(* CODESYS project SingleElevator.project

Project tree, tasks and I/O mapping:
  Device : CODESYS Control Win V3, CODESYS, version 3.5.21.30
    application Application
      libraries: Standard, 3.5.18.0 (System)
      task MainTask (cyclic, interval t#20ms, priority 1) calls Simulation, GA_collector, PLC_Program
      task VISU_TASK (cyclic, interval 100 ms, priority 31) calls VisuElems.Visu_Prg
      global variables GVL
      visualisation Visualization
      program Simulation [ST]
      data type State_FB
      data type DoWhats
      data type Action_s
      program GA_collector [FBD]
      program PLC_Program [SFC]: _astart_led_active, _ainitialize_active, _ainitialize_exit, _ago_destination_active, _ago_destination_exit, _adoors_init_active, _adoors_open_active, _adoors_init_exit, _adoors_open_exit, _adoors_open1_active, _adoors_open1_exit, _adoors_closing_exit_1, _adoors_closing_active_1, _afault_block_entry
      function block Door_opener [SFC]: _aInit_active, _aReady_active, _aReady_exit, _aopening_door_active, _aClosing_door_active, _aopening_door_exit, _afinish_closing_exit, _aopen_again_active, _aopen_again_exit, _aSetDone_active, _aSetDone_exit, _afinish_closing_active
      function block motor [SFC]: _aReady_active, _aReady_exit, _aInit_active, _adescent_active, _aascent_active, _aSetDone_active, _adeck_fault_exit, _aSetDone_exit, _amove1_active, _await1s_entry, _amove1_exit, _aSetDone1_exit, _aSetDone1_active, _astop_motor_entry, _aset_vel_active, _adummy1_entry, _aRamp_Fault_active, _aSetDone2_entry, _aSetDone2_active, _aSetDone2_exit, _aspeed_inverter_entry, _aSetDone4_active, _aSetDone4_exit, _aascent_exit, _acurrent_add_entry, _aRamp_Fault_entry
      function block LEDs [SFC]: _aAssignCalls_active, _aAssignCalls_active_1, _aInit_active, _aReady_active_1, _aReady_exit_1
  text list GlobalTextList
  function block LEDs [SFC]: _aAssignCalls_active, _aAssignCalls_active_1, _aInit_active, _aReady_active_1, _aReady_exit_1
*)

// Device/Application/State_FB
//{attribute 'qualified_only'}
//{attribute 'strict'}// if we don't comment we need to use the nameofthetype.chosentype
TYPE State_FB :
(
	S_Init := 0,// never call a variable with the same name of a step
	S_Ready:=1,
	S_Busy:=2,
	S_Faulty:=3
	// we'll use the strings so it is more readable
);
END_TYPE

// Device/Application/DoWhats
//{attribute 'qualified_only'}
//{attribute 'strict'}
TYPE DoWhats :
(
	Gotodestination := 0,
	Initialize :=1,
	door_closing:=2,
	door_opening:=3
);
END_TYPE

// Device/Application/Action_s
//{attribute 'qualified_only'}
//{attribute 'strict'}
TYPE Action_s :
(
	start_action:=0,
	Wait_comp:=1,
	setopOK:=2
);
END_TYPE

// Device/Application/GVL
{attribute 'qualified_only'}
VAR_GLOBAL
(* Elevator managing variables*)
	Open: BOOL;				(* Sensor: the door is fully open*)
	Closed: BOOL;			(* Sensor: the door is fully closed*)
	LimitDown: BOOL;		(* Sensor: lower limit sensor, if TRUE the lift has reached the lower limit*)
	LimitUp: BOOL;			(* Sensor: upper limit sensor, if TRUE the lift has reached the upper limit*)
	DeckSensor: BOOL;		(* Sensor: if TRUE the cab is in proximity of a deck*)
	RampSensor: BOOL;		(* Sensor: if TRUE the cab is in proximity of a ramp*)
	Presence :BOOL; 		(* Sensor: if TRUE something blocks the door photocell*)
	

	Closing: BOOL;			(* Actuator: if TRUE the door starts closing*)
	Opening: BOOL;			(* Actuator: the door starts opening*)
	Motor_on: BOOL;			(* Actuator: if TRUE the lift pulley motor start moving*)
	Up: BOOL;				(* Actuator parameter: if TRUE the lift moves upward, downward otherwise*)
	Vel: BOOL;				(* Actuator parameter: motor speed, if TRUE high speed, low speed otherwise*)


	Current: INT;  			(* Visualization: variable used to storage the current deck*)
    Destination: INT;		(* Visualization: variable used to storage the the destination deck*)
	

	InitialDeck: INT := 1;	(* Only for simulation: variable used to define the initial deck*)
	InitCycle: BOOL := FALSE;(* Only for simulation: used to execute the instruction at the first cycle*)
	Height: INT;			(* Only for simulation: elevator height*)
	DeckRest: INT;        	(* Only for simulation: division rest for generating deck sensor*)
	Memory: INT;
	RampRest: INT;			(* Only for simulation: division rest for generating the ramp position*)
	MemoryR: INT;
	Door: INT;				(* Only for simulation: to visualize the closing of the door*)
	Displacement: INT;		(* Only for simulation: lift displacement, dependent on the motor speed*)

 (*Inputs: internal panel variables*)
	PG: BOOL;
	P1: BOOL;
	P2: BOOL;
	P3: BOOL;
	P4: BOOL;
	P5: BOOL;
	P6: BOOL;
	P7: BOOL;

(*Visualization: internal panel variables used to turn on the LED*)
	PGVis: BOOL;
	P1Vis: BOOL;
	P2Vis: BOOL;
	P3Vis: BOOL;
	P4Vis: BOOL;
	P5Vis: BOOL;
	P6Vis: BOOL;
	P7Vis: BOOL;

(*Inputs: external panel variables*)
	UpDeckG: BOOL;
	UpDeck1: BOOL;
	UpDeck2: BOOL;
	UpDeck3: BOOL;
	UpDeck4: BOOL;
	UpDeck5: BOOL;
	UpDeck6: BOOL;
	DownDeck7: BOOL;
	DownDeck6: BOOL;
	DownDeck5: BOOL;
	DownDeck4: BOOL;
	DownDeck3: BOOL;
	DownDeck2: BOOL;
	DownDeck1: BOOL;

(*Visualization: external panel variables used to turn on the LED*)
	UpDeckGVis: BOOL;
	UpDeck1Vis: BOOL;
	UpDeck2Vis: BOOL;
	UpDeck3Vis: BOOL;
	UpDeck4Vis: BOOL;
	UpDeck5Vis: BOOL;
	UpDeck6Vis: BOOL;
	DownDeck7Vis: BOOL;
	DownDeck6Vis: BOOL;
	DownDeck5Vis: BOOL;
	DownDeck4Vis: BOOL;
	DownDeck3Vis: BOOL;
	DownDeck2Vis: BOOL;
	DownDeck1Vis: BOOL;

(*Only for simulation: variables used to simulate the fault on deck sensor*)
	SensorG: BOOL;				(* if TRUE the magnetic information for deck G is lost and the deck sensor cannot become TRUE*)
	Sensor1: BOOL;				(* if TRUE the magnetic information for deck 1 is lost and the deck sensor cannot become TRUE*)
	Sensor2: BOOL;
	Sensor3: BOOL;
	Sensor4: BOOL;
	Sensor5: BOOL;
	Sensor6: BOOL;
	Sensor7: BOOL;
	FaultSensorAlarm: BOOL; 	(* Visulaization: if TRUE alerts the user of a deck sensor fault*)

(*Only for simulation: variables used to simulate the fault on ramp sensor*)
	RampGUp: BOOL;
	Ramp1Down: BOOL;
	Ramp1Up:BOOL;
	Ramp2Down: BOOL;
	Ramp2Up:BOOL;
	Ramp3Down: BOOL;
	Ramp3Up:BOOL;
	Ramp4Down: BOOL;
	Ramp4Up:BOOL;
	Ramp5Down: BOOL;
	Ramp5Up:BOOL;
	Ramp6Down: BOOL;
	Ramp6Up:BOOL;
	Ramp7Down: BOOL;
	FaultRampAlarm: BOOL; 		(* Visulaization: if TRUE alerts the user of a ramp sensor fault*)
	SensorGOK: BOOL;
	Sensor1OK: BOOL;
	Sensor2OK: BOOL;
	Sensor6OK: BOOL;
	Sensor3OK: BOOL;
	Sensor4OK: BOOL;
	Sensor5OK: BOOL;
	Sensor7OK: BOOL;
	RampGUpOK: BOOL;
	Ramp1DownOK: BOOL;
	Ramp1UpOK: BOOL;
	Ramp2DownOK: BOOL;
	Ramp2UpOK: BOOL;
	Ramp3DownOK: BOOL;
	Ramp3UpOK: BOOL;
	Ramp4DownOK: BOOL;
	Ramp4UpOK: BOOL;
	Ramp5DownOK: BOOL;
	Ramp5UpOK: BOOL;
	Ramp6DownOK: BOOL;
	Ramp6UpOK: BOOL;
	Ramp7DownOK: BOOL;
	Ramp7UpOK: BOOL;
	Door_opener_0: Door_opener;
	motor_0: motor;
	LEDs_0: LEDs;
	state_action: Action_s;
	fault: BOOL;
END_VAR

// Device/Application/Simulation
PROGRAM Simulation
VAR
END_VAR

(* Initial position of the cab inside the hoistway. It is executed only at the first cycle.  *)
IF NOT GVL.InitCycle THEN
			GVL.InitCycle := TRUE ;
			GVL.Height := 20 * GVL.InitialDeck;
		    GVL.Door := 0;
			GVL.Current := GVL.Height / 20;
END_IF;

(* Elevator management, these instructions are executed each cycle time*)

(* Elevator door control. *)
IF GVL.Closing THEN
	GVL.Door := GVL.Door + 1;		(*Closing door management*)
	GVL.Open := FALSE;
END_IF

IF GVL.Door >= 60 THEN						(* Closed door limit*)
	GVL.Closed := TRUE;
END_IF

IF GVL.Opening THEN
	GVL.Door := GVL.Door - 1; 	(* Opening door management*)
	GVL.Closed := FALSE;
END_IF

IF GVL.Door <= 0 THEN							(* Open door limit*)
	GVL.Open := TRUE;
END_IF


(* Maximum and minimum management in the door simulation*)
IF GVL.Door < 0 THEN
	 GVL.Door := 0;
END_IF

IF GVL.Door > 60 THEN
	GVL.Door := 60;
END_IF


(* Control of the cab position inside the hostway. *)
(* Displacement definition for graphic visualization*)
IF GVL.Vel THEN 
	GVL.Displacement := 2;
ELSE 
	GVL.Displacement := 1;
END_IF


(* Height modification relying on direction and speed*)
IF GVL.Motor_on AND GVL.Up THEN
	GVL.Height := GVL.Height + GVL.Displacement;
	GVL.LimitDown := FALSE;
END_IF

IF GVL.Motor_on AND NOT GVL.Up THEN
	GVL.Height := GVL.Height - GVL.Displacement;
	GVL.LimitUp := FALSE;
END_IF


(* Limits for visualization*)
IF GVL.Height < -20 THEN
	GVL.Height := -20;
END_IF

IF GVL.Height > 160 THEN
	GVL.Height := 160;
END_IF

(* Limit sensors management*)
IF GVL.Height <= -10 THEN
	GVL.LimitDown := TRUE;
END_IF

IF GVL.Height >= 150 THEN
	 GVL.LimitUp := TRUE;
END_IF


(*-------------------------------------------------------------------*)
(*  Fault Management (Deck and Ramp Sensors)   *)
(*-------------------------------------------------------------------*)
(* Deck Sensor*)
(* Range of value where the deck sensor is active*)
IF ((GVL.Height >= -1) AND (GVL.Height <= 1)) THEN
	GVL.SensorGOK := TRUE;
ELSE  
	GVL.SensorGOK := FALSE;
END_IF

IF ((GVL.Height >= 20-1) AND (GVL.Height <= 20+1)) THEN
	GVL.Sensor1OK := TRUE;
ELSE  
	GVL.Sensor1OK := FALSE;
END_IF

IF ((GVL.Height >= 40-1) AND (GVL.Height <= 40+1)) THEN
	GVL.Sensor2OK := TRUE;
ELSE  
	GVL.Sensor2OK := FALSE;
END_IF

IF ((GVL.Height >= 60-1) AND (GVL.Height <= 60+1)) THEN
	GVL.Sensor3OK := TRUE;
ELSE  
	GVL.Sensor3OK := FALSE;
END_IF

IF ((GVL.Height >= 80-1) AND (GVL.Height <= 80+1)) THEN
	GVL.Sensor4OK := TRUE;
ELSE  
	GVL.Sensor4OK := FALSE;
END_IF

IF ((GVL.Height >= 100-1) AND (GVL.Height <= 100+1)) THEN
	GVL.Sensor5OK := TRUE;
ELSE   
	GVL.Sensor5OK := FALSE;
END_IF

IF ((GVL.Height >= 120-1) AND (GVL.Height <= 120+1)) THEN
	GVL.Sensor6OK := TRUE;
ELSE  
	GVL.Sensor6OK := FALSE;
END_IF

IF ((GVL.Height >= 140-1) AND (GVL.Height <= 140+1)) THEN
	GVL.Sensor7OK := TRUE;
ELSE  
	GVL.Sensor7OK := FALSE;
END_IF

GVL.DeckSensor := (GVL.SensorGOK AND NOT GVL.SensorG) OR
				    (GVL.Sensor1OK AND NOT GVL.Sensor1) OR
				    (GVL.Sensor2OK AND NOT GVL.Sensor2) OR
				    (GVL.Sensor3OK AND NOT GVL.Sensor3) OR
				    (GVL.Sensor4OK AND NOT GVL.Sensor4) OR
				    (GVL.Sensor5OK AND NOT GVL.Sensor5) OR
				    (GVL.Sensor6OK AND NOT GVL.Sensor6) OR
				    (GVL.Sensor7OK AND NOT GVL.Sensor7);

(* Ramp Sensor*)
(* Range of value where the ramp sensor is active*)
IF ((GVL.Height >= 5-1) AND (GVL.Height <= 5+1)) THEN
	GVL.RampGUpOK := TRUE;
ELSE 
	GVL.RampGUpOK := FALSE;
END_IF

(* Ramp close to deck 1*)
IF ((GVL.Height >= 15-1) AND (GVL.Height <= 15+1)) THEN
	GVL.Ramp1DownOK := TRUE;
ELSE 
	GVL.Ramp1DownOK := FALSE;
END_IF

IF ((GVL.Height >= 25-1) AND (GVL.Height <= 25+1)) THEN
	GVL.Ramp1UpOK := TRUE;
ELSE 
	GVL.Ramp1UpOK := FALSE;
END_IF

(* Ramp close to deck 2*)
IF ((GVL.Height >= 35-1) AND (GVL.Height <= 35+1)) THEN
	GVL.Ramp2DownOK := TRUE;
ELSE 
	GVL.Ramp2DownOK := FALSE;
END_IF

IF ((GVL.Height >= 45-1) AND (GVL.Height <= 45+1)) THEN
	GVL.Ramp2UpOK := TRUE;
ELSE 
	GVL.Ramp2UpOK := FALSE;
END_IF

(*Ramp close to deck  3*)
IF ((GVL.Height >= 55-1) AND (GVL.Height <= 55+1)) THEN
	GVL.Ramp3DownOK := TRUE;
ELSE 
	GVL.Ramp3DownOK := FALSE;
END_IF

IF ((GVL.Height >= 65-1) AND (GVL.Height <= 65+1)) THEN
	GVL.Ramp3UpOK := TRUE;
ELSE 
	GVL.Ramp3UpOK := FALSE;
END_IF

(* Ramp close to deck  4*)
IF ((GVL.Height >= 75-1) AND (GVL.Height <= 75+1)) THEN
	GVL.Ramp4DownOK := TRUE;
ELSE 
	GVL.Ramp4DownOK := FALSE;
END_IF

IF ((GVL.Height >= 85-1) AND (GVL.Height <= 85+1)) THEN
	GVL.Ramp4UpOK := TRUE;
ELSE 
	GVL.Ramp4UpOK:=FALSE;
END_IF

(* Ramp close to deck  5*)
IF ((GVL.Height >= 95-1) AND (GVL.Height <= 95+1)) THEN
	GVL.Ramp5DownOK := TRUE;
ELSE 
	GVL.Ramp5DownOK := FALSE;
END_IF

IF ((GVL.Height >= 105-1) AND (GVL.Height <= 105+1)) THEN
	GVL.Ramp5UpOK := TRUE;
ELSE
	GVL.Ramp5UpOK := FALSE;
END_IF

(* Ramp close to deck  6*)
IF ((GVL.Height >= 115-1) AND (GVL.Height <= 115+1)) THEN
	GVL.Ramp6DownOK := TRUE;
ELSE 
	GVL.Ramp6DownOK := FALSE;
END_IF

IF ((GVL.Height >= 125-1) AND (GVL.Height <= 125+1)) THEN
	GVL.Ramp6UpOK := TRUE;
ELSE 
	GVL.Ramp6UpOK := FALSE;
END_IF

(* Ramp close to deck  7*)
IF ((GVL.Height >= 135-1) AND (GVL.Height <= 135+1)) THEN
	GVL.Ramp7DownOK := TRUE;
ELSE 
	GVL.Ramp7DownOK := FALSE;
END_IF

GVL.RampSensor:=(GVL.RampGUpOK AND NOT GVL.RampGUp) OR 
								(GVL.Ramp1DownOK AND NOT GVL.Ramp1Down ) OR 
								(GVL.Ramp1UpOK AND NOT GVL.Ramp1Up ) OR
								(GVL.Ramp2DownOK AND NOT GVL.Ramp2Down ) OR 
								(GVL.Ramp2UpOK AND NOT GVL.Ramp2Up ) OR
								(GVL.Ramp3DownOK AND NOT GVL.Ramp3Down ) OR
 								(GVL.Ramp3UpOK AND NOT GVL.Ramp3Up ) OR
								(GVL.Ramp4DownOK AND NOT GVL.Ramp4Down ) OR
 								(GVL.Ramp4UpOK AND NOT GVL.Ramp4Up ) OR
								(GVL.Ramp5DownOK AND NOT GVL.Ramp5Down ) OR
 								(GVL.Ramp5UpOK AND NOT GVL.Ramp5Up ) OR
								(GVL.Ramp6DownOK AND NOT GVL.Ramp6Down ) OR
								(GVL.Ramp6UpOK AND NOT GVL.Ramp6Up ) OR
								(GVL.Ramp7DownOK AND NOT GVL.Ramp7Down );

END_PROGRAM

// Device/Application/GA_collector
PROGRAM GA_collector
VAR
END_VAR

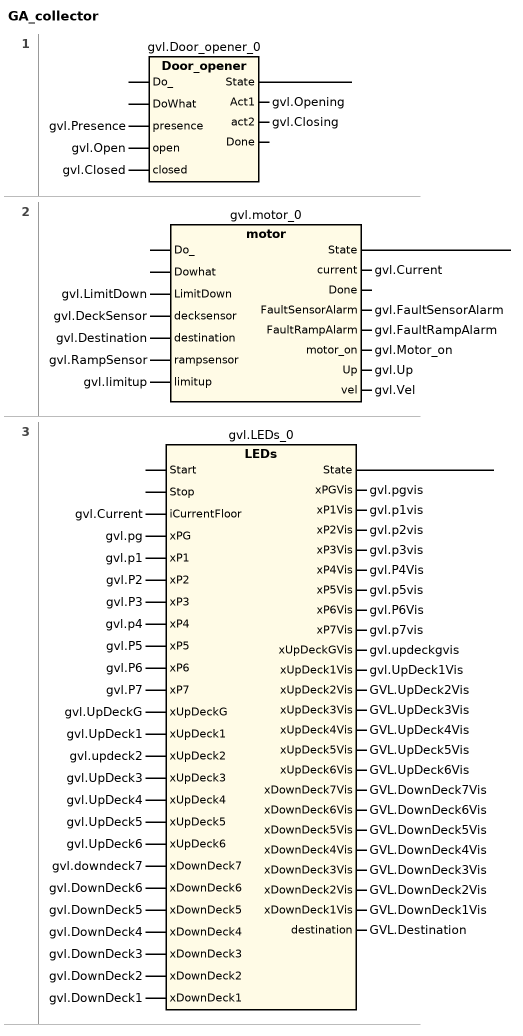
// NETWORK 1
gvl.Door_opener_0(
    presence := gvl.Presence,
    open := gvl.Open,
    closed := gvl.Closed,
    Act1 => gvl.Opening,
    act2 => gvl.Closing); // Door_opener

// NETWORK 2
gvl.motor_0(
    LimitDown := gvl.LimitDown,
    decksensor := gvl.DeckSensor,
    destination := gvl.Destination,
    rampsensor := gvl.RampSensor,
    limitup := gvl.limitup,
    current => gvl.Current,
    FaultSensorAlarm => gvl.FaultSensorAlarm,
    FaultRampAlarm => gvl.FaultRampAlarm,
    motor_on => gvl.Motor_on,
    Up => gvl.Up,
    vel => gvl.Vel); // motor

// NETWORK 3
gvl.LEDs_0(
    iCurrentFloor := gvl.Current,
    xPG := gvl.pg,
    xP1 := gvl.p1,
    xP2 := gvl.P2,
    xP3 := gvl.P3,
    xP4 := gvl.p4,
    xP5 := gvl.P5,
    xP6 := gvl.P6,
    xP7 := gvl.P7,
    xUpDeckG := gvl.UpDeckG,
    xUpDeck1 := gvl.UpDeck1,
    xUpDeck2 := gvl.updeck2,
    xUpDeck3 := gvl.UpDeck3,
    xUpDeck4 := gvl.UpDeck4,
    xUpDeck5 := gvl.UpDeck5,
    xUpDeck6 := gvl.UpDeck6,
    xDownDeck7 := gvl.downdeck7,
    xDownDeck6 := gvl.DownDeck6,
    xDownDeck5 := gvl.DownDeck5,
    xDownDeck4 := gvl.DownDeck4,
    xDownDeck3 := gvl.DownDeck3,
    xDownDeck2 := gvl.DownDeck2,
    xDownDeck1 := gvl.DownDeck1,
    xPGVis => gvl.pgvis,
    xP1Vis => gvl.p1vis,
    xP2Vis => gvl.p2vis,
    xP3Vis => gvl.p3vis,
    xP4Vis => gvl.P4Vis,
    xP5Vis => gvl.p5vis,
    xP6Vis => gvl.P6Vis,
    xP7Vis => gvl.p7vis,
    xUpDeckGVis => gvl.updeckgvis,
    xUpDeck1Vis => gvl.UpDeck1Vis,
    xUpDeck2Vis => GVL.UpDeck2Vis,
    xUpDeck3Vis => GVL.UpDeck3Vis,
    xUpDeck4Vis => GVL.UpDeck4Vis,
    xUpDeck5Vis => GVL.UpDeck5Vis,
    xUpDeck6Vis => GVL.UpDeck6Vis,
    xDownDeck7Vis => GVL.DownDeck7Vis,
    xDownDeck6Vis => GVL.DownDeck6Vis,
    xDownDeck5Vis => GVL.DownDeck5Vis,
    xDownDeck4Vis => GVL.DownDeck4Vis,
    xDownDeck3Vis => GVL.DownDeck3Vis,
    xDownDeck2Vis => GVL.DownDeck2Vis,
    xDownDeck1Vis => GVL.DownDeck1Vis,
    destination => GVL.Destination); // LEDs

END_PROGRAM

// Device/Application/Door_opener
FUNCTION_BLOCK Door_opener
VAR_INPUT
	Do_: BOOL;
	DoWhat: DoWhats;
	presence: BOOL;
	open: BOOL;
	closed: BOOL;
END_VAR
VAR_OUTPUT
	State: STATE_FB;
	Act1: BOOL;
	act2: BOOL;
	Done: BOOL;
END_VAR
VAR
END_VAR

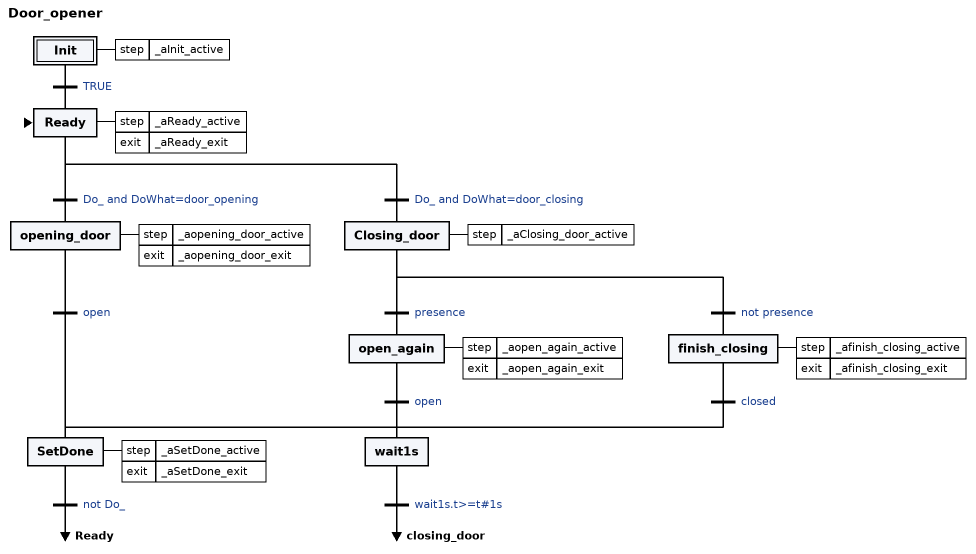
INITIAL_STEP Init:
    _aInit_active(N);  // step action
END_STEP
TRANSITION FROM Init TO Ready
    := TRUE;
END_TRANSITION
STEP Ready:
    _aReady_active(N);  // step action
    _aReady_exit(P0);  // exit action
END_STEP
TRANSITION FROM Ready TO opening_door
    := Do_ and DoWhat=door_opening;
END_TRANSITION
STEP opening_door:
    _aopening_door_active(N);  // step action
    _aopening_door_exit(P0);  // exit action
END_STEP
TRANSITION FROM opening_door TO SetDone
    := open;
END_TRANSITION
TRANSITION FROM Ready TO Closing_door
    := Do_ and DoWhat=door_closing;
END_TRANSITION
STEP Closing_door:
    _aClosing_door_active(N);  // step action
END_STEP
TRANSITION FROM Closing_door TO open_again
    := presence;
END_TRANSITION
STEP open_again:
    _aopen_again_active(N);  // step action
    _aopen_again_exit(P0);  // exit action
END_STEP
TRANSITION FROM open_again TO wait1s
    := open;
END_TRANSITION
STEP wait1s:
END_STEP
TRANSITION FROM wait1s TO closing_door
    := wait1s.t>=t#1s;
END_TRANSITION
TRANSITION FROM Closing_door TO finish_closing
    := not presence;
END_TRANSITION
STEP finish_closing:
    _afinish_closing_active(N);  // step action
    _afinish_closing_exit(P0);  // exit action
END_STEP
TRANSITION FROM finish_closing TO SetDone
    := closed;
END_TRANSITION
STEP SetDone:
    _aSetDone_active(N);  // step action
    _aSetDone_exit(P0);  // exit action
END_STEP
TRANSITION FROM SetDone TO Ready
    := not Do_;
END_TRANSITION

ACTION _aInit_active:
State := S_init;
END_ACTION

ACTION _aReady_active:
state:=S_ready;
END_ACTION

ACTION _aReady_exit:
state:=S_busy;
END_ACTION

ACTION _aopening_door_active:
Act1:=true;
END_ACTION

ACTION _aClosing_door_active:
IF NOT presence THEN
	act2:=TRUE;
END_IF
END_ACTION

ACTION _aopening_door_exit:
Act1:=FALSE;
END_ACTION

ACTION _afinish_closing_exit:
Act2:=FALSE;
END_ACTION

ACTION _aopen_again_active:
act1:=true;
END_ACTION

ACTION _aopen_again_exit:
act1:=false;
END_ACTION

ACTION _aSetDone_active:
Done:=TRUE;
END_ACTION

ACTION _aSetDone_exit:
Done:=false;
END_ACTION

ACTION _afinish_closing_active:
IF presence THEN
	act2:=FALSE;
	act1:=TRUE;
	IF open AND NOT presence THEN
		act1:=FALSE;
		act2:=TRUE;
	END_IF
END_IF
IF NOT presence THEN
		act1:=FALSE;
		act2:=TRUE;
END_IF
END_ACTION

END_FUNCTION_BLOCK

// Device/Application/motor
FUNCTION_BLOCK motor
VAR_INPUT
	Do_: BOOL;
	Dowhat: DoWhats;
	LimitDown: BOOL;
	decksensor: BOOL;
	destination: INT;  //DESTINAZIONI;
	rampsensor: BOOL;
	limitup: BOOL;
END_VAR
VAR_OUTPUT
	State: STATE_FB;
	current: INT;//destinazioni;
	Done: BOOL;
	FaultSensorAlarm: BOOL;
	FaultRampAlarm: BOOL;
	motor_on: BOOL;
	Up: BOOL;
	vel: BOOL;
END_VAR
VAR
	num_ramp: INT;
	destination_mem: INT;
END_VAR

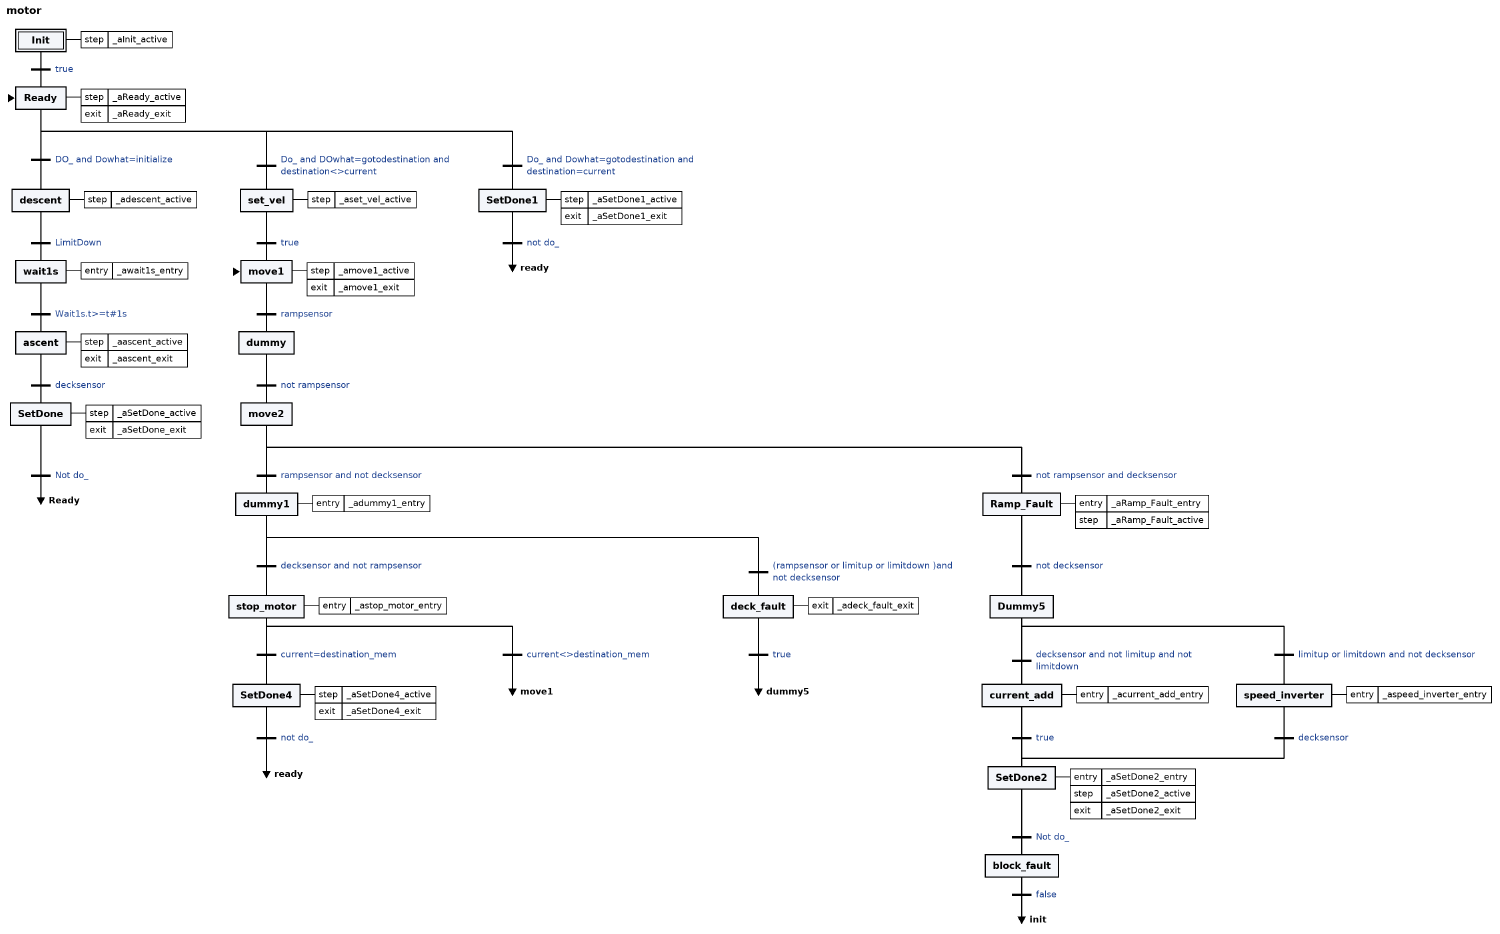
INITIAL_STEP Init:
    _aInit_active(N);  // step action
END_STEP
TRANSITION FROM Init TO Ready
    := true;
END_TRANSITION
STEP Ready:
    _aReady_active(N);  // step action
    _aReady_exit(P0);  // exit action
END_STEP
TRANSITION FROM Ready TO descent
    := DO_ and Dowhat=initialize;
END_TRANSITION
STEP descent:
    _adescent_active(N);  // step action
END_STEP
TRANSITION FROM descent TO wait1s
    := LimitDown;
END_TRANSITION
STEP wait1s:
    _await1s_entry(P1);  // entry action
END_STEP
TRANSITION FROM wait1s TO ascent
    := Wait1s.t>=t#1s;
END_TRANSITION
STEP ascent:
    _aascent_active(N);  // step action
    _aascent_exit(P0);  // exit action
END_STEP
TRANSITION FROM ascent TO SetDone
    := decksensor;
END_TRANSITION
STEP SetDone:
    _aSetDone_active(N);  // step action
    _aSetDone_exit(P0);  // exit action
END_STEP
TRANSITION FROM SetDone TO Ready
    := Not do_;
END_TRANSITION
TRANSITION FROM Ready TO set_vel
    := Do_ and DOwhat=gotodestination and destination<>current;
END_TRANSITION
STEP set_vel:
    _aset_vel_active(N);  // step action
END_STEP
TRANSITION FROM set_vel TO move1
    := true;
END_TRANSITION
STEP move1:
    _amove1_active(N);  // step action
    _amove1_exit(P0);  // exit action
END_STEP
TRANSITION FROM move1 TO dummy
    := rampsensor;
END_TRANSITION
STEP dummy:
END_STEP
TRANSITION FROM dummy TO move2
    := not rampsensor;
END_TRANSITION
STEP move2:
END_STEP
TRANSITION FROM move2 TO dummy1
    := rampsensor and not decksensor;
END_TRANSITION
STEP dummy1:
    _adummy1_entry(P1);  // entry action
END_STEP
TRANSITION FROM dummy1 TO stop_motor
    := decksensor and not rampsensor;
END_TRANSITION
STEP stop_motor:
    _astop_motor_entry(P1);  // entry action
END_STEP
TRANSITION FROM dummy1 TO deck_fault
    := (rampsensor or limitup or limitdown )and not decksensor;
END_TRANSITION
STEP deck_fault:
    _adeck_fault_exit(P0);  // exit action
END_STEP
TRANSITION FROM deck_fault TO dummy5
    := true;
END_TRANSITION
TRANSITION FROM stop_motor TO SetDone4
    := current=destination_mem;
END_TRANSITION
STEP SetDone4:
    _aSetDone4_active(N);  // step action
    _aSetDone4_exit(P0);  // exit action
END_STEP
TRANSITION FROM SetDone4 TO ready
    := not do_;
END_TRANSITION
TRANSITION FROM stop_motor TO move1
    := current<>destination_mem;
END_TRANSITION
TRANSITION FROM move2 TO Ramp_Fault
    := not rampsensor and decksensor;
END_TRANSITION
STEP Ramp_Fault:
    _aRamp_Fault_entry(P1);  // entry action
    _aRamp_Fault_active(N);  // step action
END_STEP
TRANSITION FROM Ramp_Fault TO Dummy5
    := not decksensor;
END_TRANSITION
STEP Dummy5:
END_STEP
TRANSITION FROM Dummy5 TO current_add
    := decksensor and not limitup and not limitdown;
END_TRANSITION
STEP current_add:
    _acurrent_add_entry(P1);  // entry action
END_STEP
TRANSITION FROM current_add TO SetDone2
    := true;
END_TRANSITION
TRANSITION FROM Dummy5 TO speed_inverter
    := limitup or limitdown and not decksensor;
END_TRANSITION
STEP speed_inverter:
    _aspeed_inverter_entry(P1);  // entry action
END_STEP
TRANSITION FROM speed_inverter TO SetDone2
    := decksensor;
END_TRANSITION
STEP SetDone2:
    _aSetDone2_entry(P1);  // entry action
    _aSetDone2_active(N);  // step action
    _aSetDone2_exit(P0);  // exit action
END_STEP
TRANSITION FROM SetDone2 TO block_fault
    := Not do_;
END_TRANSITION
STEP block_fault:
END_STEP
TRANSITION FROM block_fault TO init
    := false;
END_TRANSITION
TRANSITION FROM Ready TO SetDone1
    := Do_ and Dowhat=gotodestination and destination=current;
END_TRANSITION
STEP SetDone1:
    _aSetDone1_active(N);  // step action
    _aSetDone1_exit(P0);  // exit action
END_STEP
TRANSITION FROM SetDone1 TO ready
    := not do_;
END_TRANSITION

ACTION _aReady_active:
State:= S_Ready;
END_ACTION

ACTION _aReady_exit:
State:= S_Busy;
END_ACTION

ACTION _aInit_active:
state:= S_init;
END_ACTION

ACTION _adescent_active:
motor_on:=TRUE;
Up:=FALSE;
vel:=FALSE;
END_ACTION

ACTION _aascent_active:
motor_on:=TRUE;
up:=TRUE;
vel:=FALSE;
current:=0; //1;
END_ACTION

ACTION _aSetDone_active:
Done:= TRUE;
END_ACTION

ACTION _adeck_fault_exit:
FaultSensorAlarm:=TRUE;
vel:=False;
END_ACTION

ACTION _aSetDone_exit:
Done:=FALSE;
END_ACTION

ACTION _amove1_active:
IF destination>current THEN
motor_on:=TRUE;
up:=TRUE;
num_ramp:=2*(destination-current);
END_IF

IF destination<current THEN
motor_on:=TRUE;
up:=FALSE;
num_ramp:=2*(current-destination);
END_IF
END_ACTION

ACTION _await1s_entry:
motor_on:=false;
END_ACTION

ACTION _amove1_exit:
vel:=true;
END_ACTION

ACTION _aSetDone1_exit:
Done:=FALSE;
END_ACTION

ACTION _aSetDone1_active:
Done:= TRUE;
motor_on:=false;
END_ACTION

ACTION _astop_motor_entry:
IF current=destination_mem THEN
	motor_on:=FALSE;
END_IF
END_ACTION

ACTION _aset_vel_active:
vel:=FALSE;
END_ACTION

ACTION _adummy1_entry:
IF destination=-1 THEN
	destination_mem:=0;
	ELSE
	destination_mem:=destination;
END_IF


IF up=TRUE THEN
current:=current +1;
END_IF

IF up=FALSE THEN
current:=current -1;
END_IF

IF current=destination THEN
	vel:=FALSE;
END_IF
END_ACTION

ACTION _aRamp_Fault_active:
FaultRampAlarm:=TRUE;
Vel:=FALSE;
END_ACTION

ACTION _aSetDone2_entry:
motor_on:=false;
END_ACTION

ACTION _aSetDone2_active:
Done:=TRUE;
State:=3;
END_ACTION

ACTION _aSetDone2_exit:
Done:=false;
END_ACTION

ACTION _aspeed_inverter_entry:
up:= NOT up;

IF up=TRUE THEN
	IF faultrampalarm=1 THEN
		current:=0;
	END_IF
	IF faultrampalarm=0 THEN
		current:=1;
	END_IF;
END_IF

IF up=FALSE THEN
		IF faultrampalarm=1 THEN
		current:=7;
	END_IF
	IF faultrampalarm=0 THEN
		current:=6;
	END_IF;
END_IF
END_ACTION

ACTION _aSetDone4_active:
Done:= TRUE;
END_ACTION

ACTION _aSetDone4_exit:
Done:=FALSE;
END_ACTION

ACTION _aascent_exit:
motor_on:=false;
END_ACTION

ACTION _acurrent_add_entry:
IF up=TRUE THEN
current:=current +1;
END_IF

IF up=FALSE THEN
current:=current -1;
END_IF
END_ACTION

ACTION _aRamp_Fault_entry:
IF up=TRUE THEN
current:=current +1;
END_IF

IF up=FALSE THEN
current:=current -1;
END_IF
END_ACTION

END_FUNCTION_BLOCK

// LEDs
FUNCTION_BLOCK LEDs
VAR_INPUT
	Start: BOOL;
	Stop: BOOL;
	iCurrentFloor:INT;
	xPG: BOOL;
	xP1: BOOL;
	xP2: BOOL;
	xP3: BOOL;
	xP4: BOOL;
	xP5: BOOL;
	xP6: BOOL;
	xP7: BOOL;
	xUpDeckG: BOOL;
	xUpDeck1: BOOL;
	xUpDeck2: BOOL;
	xUpDeck3: BOOL;
	xUpDeck4: BOOL;
	xUpDeck5: BOOL;
	xUpDeck6: BOOL;
	xDownDeck7: BOOL;
	xDownDeck6: BOOL;
	xDownDeck5: BOOL;
	xDownDeck4: BOOL;
	xDownDeck3: BOOL;
	xDownDeck2: BOOL;
	xDownDeck1: BOOL;
END_VAR
VAR_OUTPUT
	State: STATE_FB;
	//arrCalls: ARRAY [0..7] OF BOOL;
	xPGVis: BOOL;
	xP1Vis: BOOL;
	xP2Vis: BOOL;
	xP3Vis: BOOL;
	xP4Vis: BOOL;
	xP5Vis: BOOL;
	xP6Vis: BOOL;
	xP7Vis: BOOL;
	xUpDeckGVis: BOOL;
	xUpDeck1Vis: BOOL;
	xUpDeck2Vis: BOOL;
	xUpDeck3Vis: BOOL;
	xUpDeck4Vis: BOOL;
	xUpDeck5Vis: BOOL;
	xUpDeck6Vis: BOOL;
	xDownDeck7Vis: BOOL;
	xDownDeck6Vis: BOOL;
	xDownDeck5Vis: BOOL;
	xDownDeck4Vis: BOOL;
	xDownDeck3Vis: BOOL;
	xDownDeck2Vis: BOOL;
	xDownDeck1Vis: BOOL;
	destination:INT;
END_VAR
VAR
	arrButtons : ARRAY [0..7] OF BOOL;
	i: INT:=0;
	k: INT;
	destinations : ARRAY [0..7] OF INT;
	skip: BOOL;
	z: INT := 0;
	w: INT :=0;
	y: INT := 0;
	q: INT := 0;
END_VAR

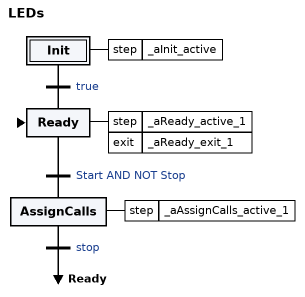
INITIAL_STEP Init:
    _aInit_active(N);  // step action
END_STEP
TRANSITION FROM Init TO Ready
    := true;
END_TRANSITION
STEP Ready:
    _aReady_active_1(N);  // step action
    _aReady_exit_1(P0);  // exit action
END_STEP
TRANSITION FROM Ready TO AssignCalls
    := Start AND NOT Stop;
END_TRANSITION
STEP AssignCalls:
    _aAssignCalls_active_1(N);  // step action
END_STEP
TRANSITION FROM AssignCalls TO Ready
    := stop;
END_TRANSITION

ACTION _aAssignCalls_active:
arrButtons[0]:= (xPG OR xUpDeckG);
arrButtons[1]:= (xP1 OR xUpDeck1 OR xDownDeck1);
arrButtons[2]:= (xP2 OR xUpDeck2 OR xDownDeck2);
arrButtons[3]:= (xP3 OR xUpDeck3 OR xDownDeck3);
arrButtons[4]:= (xP4 OR xUpDeck4 OR xDownDeck4);
arrButtons[5]:= (xP5 OR xUpDeck5 OR xDownDeck5);
arrButtons[6]:= (xP6 OR xUpDeck6 OR xDownDeck6);
arrButtons[7]:= (xP7 OR xDownDeck7);
END_ACTION

ACTION _aAssignCalls_active_1:
IF xPG OR xUpDeckG THEN
arrButtons[0]:= (xPG OR xUpDeckG);
END_IF
IF (xP1 OR xUpDeck1 OR xDownDeck1) THEN
arrButtons[1]:= (xP1 OR xUpDeck1 OR xDownDeck1);
END_IF
IF (xP2 OR xUpDeck2 OR xDownDeck2) THEN
arrButtons[2]:= (xP2 OR xUpDeck2 OR xDownDeck2);
END_IF
IF (xP3 OR xUpDeck3 OR xDownDeck3) THEN
arrButtons[3]:= (xP3 OR xUpDeck3 OR xDownDeck3);
END_IF
IF (xP4 OR xUpDeck4 OR xDownDeck4) THEN
arrButtons[4]:= (xP4 OR xUpDeck4 OR xDownDeck4);
END_IF
IF (xP5 OR xUpDeck5 OR xDownDeck5) THEN
arrButtons[5]:= (xP5 OR xUpDeck5 OR xDownDeck5);
END_IF
IF (xP6 OR xUpDeck6 OR xDownDeck6) THEN
arrButtons[6]:= (xP6 OR xUpDeck6 OR xDownDeck6);
END_IF
IF (xP7 OR xDownDeck7) THEN
arrButtons[7]:= (xP7 OR xDownDeck7);
END_IF

FOR z:= 0 TO 7 DO
	IF arrbuttons[z]=1 THEN
		//accensione luci pulsanti
		//se un certo pulsante è chiamato accendi la relativa luce
		
//pulsanti pannello interno
		IF xPG = 1 THEN xPGVis := 1; END_IF
		IF xP1 = 1 THEN xP1Vis := 1; END_IF
		IF xP2 = 1 THEN xP2Vis := 1; END_IF
		IF xP3 = 1 THEN xP3Vis := 1; END_IF
		IF xP4 = 1 THEN xP4Vis := 1; END_IF
		IF xP5 = 1 THEN xP5Vis := 1; END_IF
		IF xP6 = 1 THEN xP6Vis := 1; END_IF
		IF xP7 = 1 THEN xP7Vis := 1; END_IF
//pulsanti UpDeck
		IF xUpDeckG = 1 THEN xUpDeckGVis := 1; END_IF
		IF xUpDeck1 = 1 THEN xUpDeck1Vis := 1; END_IF
		IF xUpDeck2 = 1 THEN xUpDeck2Vis := 1; END_IF
		IF xUpDeck3 = 1 THEN xUpDeck3Vis := 1; END_IF
		IF xUpDeck4 = 1 THEN xUpDeck4Vis := 1; END_IF
		IF xUpDeck5 = 1 THEN xUpDeck5Vis := 1; END_IF
		IF xUpDeck6 = 1 THEN xUpDeck6Vis := 1; END_IF
//pulsanti DownDeck
		IF xDownDeck1 = 1 THEN xDownDeck1Vis := 1; END_IF
		IF xDownDeck2 = 1 THEN xDownDeck2Vis := 1; END_IF
		IF xDownDeck3 = 1 THEN xDownDeck3Vis := 1; END_IF
		IF xDownDeck4 = 1 THEN xDownDeck4Vis := 1; END_IF
		IF xDownDeck5 = 1 THEN xDownDeck5Vis := 1; END_IF
		IF xDownDeck6 = 1 THEN xDownDeck6Vis := 1; END_IF
		IF xDownDeck7 = 1 THEN xDownDeck7Vis := 1; END_IF
		
		//assegna le chiamate nelle destinazioni
		skip := FALSE; //inizializza skip a ogni giro
		FOR k :=0 TO 7 DO
			IF destinations[k]=z THEN //se c'è gia una chiamata
				arrbuttons[z]:=0;
				skip := TRUE;
			END_IF 
			IF (destinations[k]=-1 AND NOT skip) THEN 
					destinations[k]:=z;	//assegna la chiamata
					EXIT;

			END_IF	
		END_FOR
		//le luci sono state accese
		//le chiamate assegnate
		//e controllato se c'erano doppioni
		destination:= destinations[0];
	END_IF
END_FOR




//spegni luci
    IF iCurrentFloor = destination THEN
		CASE iCurrentFloor OF
			0:
 				xPGVis := FALSE;
				xUpDeckGVis := FALSE;
  			1:  
        		xP1Vis := FALSE;       
        		xUpDeck1Vis := FALSE;   
       			xDownDeck1Vis := FALSE;
			2:  
        		xP2Vis := FALSE;       
        		xUpDeck2Vis := FALSE;   
       			xDownDeck2Vis := FALSE;
			3:  
        		xP3Vis := FALSE;       
        		xUpDeck3Vis := FALSE;   
       			xDownDeck3Vis := FALSE;
			4:  
        		xP4Vis := FALSE;       
        		xUpDeck2Vis := FALSE;   
       			xDownDeck2Vis := FALSE;
			5:  
        		xP5Vis := FALSE;       
        		xUpDeck5Vis := FALSE;   
       			xDownDeck5Vis := FALSE;
			6:  
        		xP6Vis := FALSE;       
        		xUpDeck6Vis := FALSE;   
       			xDownDeck6Vis := FALSE;
			7:  
        		xP7Vis := FALSE;        
       			xDownDeck7Vis := FALSE;		
		END_CASE
		
		FOR w := 0 TO 6 DO
        	Destinations[w] := Destinations[w + 1];
    	END_FOR;
		
		destinations[7]:=-1;
		destination:=destinations[0];
		
    END_IF
END_ACTION

ACTION _aInit_active:
State:=S_init;
FOR y:=0 TO 7 DO
	Destinations[y] := -1; 
END_FOR
END_ACTION

ACTION _aReady_active_1:
State:=S_ready;
END_ACTION

ACTION _aReady_exit_1:
state:=S_busy;
END_ACTION

END_FUNCTION_BLOCK

// Device/Application/LEDs
FUNCTION_BLOCK LEDs
VAR_INPUT
	Start: BOOL;
	Stop: BOOL;
	iCurrentFloor:INT;
	xPG: BOOL;
	xP1: BOOL;
	xP2: BOOL;
	xP3: BOOL;
	xP4: BOOL;
	xP5: BOOL;
	xP6: BOOL;
	xP7: BOOL;
	xUpDeckG: BOOL;
	xUpDeck1: BOOL;
	xUpDeck2: BOOL;
	xUpDeck3: BOOL;
	xUpDeck4: BOOL;
	xUpDeck5: BOOL;
	xUpDeck6: BOOL;
	xDownDeck7: BOOL;
	xDownDeck6: BOOL;
	xDownDeck5: BOOL;
	xDownDeck4: BOOL;
	xDownDeck3: BOOL;
	xDownDeck2: BOOL;
	xDownDeck1: BOOL;
END_VAR
VAR_OUTPUT
	State: STATE_FB;
	//arrCalls: ARRAY [0..7] OF BOOL;
	xPGVis: BOOL;
	xP1Vis: BOOL;
	xP2Vis: BOOL;
	xP3Vis: BOOL;
	xP4Vis: BOOL;
	xP5Vis: BOOL;
	xP6Vis: BOOL;
	xP7Vis: BOOL;
	xUpDeckGVis: BOOL;
	xUpDeck1Vis: BOOL;
	xUpDeck2Vis: BOOL;
	xUpDeck3Vis: BOOL;
	xUpDeck4Vis: BOOL;
	xUpDeck5Vis: BOOL;
	xUpDeck6Vis: BOOL;
	xDownDeck7Vis: BOOL;
	xDownDeck6Vis: BOOL;
	xDownDeck5Vis: BOOL;
	xDownDeck4Vis: BOOL;
	xDownDeck3Vis: BOOL;
	xDownDeck2Vis: BOOL;
	xDownDeck1Vis: BOOL;
	destination:INT;
END_VAR
VAR
	arrButtons : ARRAY [0..7] OF BOOL;
	i: INT:=0;
	k: INT;
	destinations : ARRAY [0..7] OF INT;
	skip: BOOL;
	z: INT := 0;
	w: INT :=0;
	y: INT := 0;
	q: INT := 0;
END_VAR

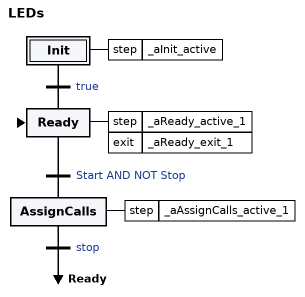
INITIAL_STEP Init:
    _aInit_active(N);  // step action
END_STEP
TRANSITION FROM Init TO Ready
    := true;
END_TRANSITION
STEP Ready:
    _aReady_active_1(N);  // step action
    _aReady_exit_1(P0);  // exit action
END_STEP
TRANSITION FROM Ready TO AssignCalls
    := Start AND NOT Stop;
END_TRANSITION
STEP AssignCalls:
    _aAssignCalls_active_1(N);  // step action
END_STEP
TRANSITION FROM AssignCalls TO Ready
    := stop;
END_TRANSITION

ACTION _aAssignCalls_active:
arrButtons[0]:= (xPG OR xUpDeckG);
arrButtons[1]:= (xP1 OR xUpDeck1 OR xDownDeck1);
arrButtons[2]:= (xP2 OR xUpDeck2 OR xDownDeck2);
arrButtons[3]:= (xP3 OR xUpDeck3 OR xDownDeck3);
arrButtons[4]:= (xP4 OR xUpDeck4 OR xDownDeck4);
arrButtons[5]:= (xP5 OR xUpDeck5 OR xDownDeck5);
arrButtons[6]:= (xP6 OR xUpDeck6 OR xDownDeck6);
arrButtons[7]:= (xP7 OR xDownDeck7);
END_ACTION

ACTION _aAssignCalls_active_1:
IF xPG OR xUpDeckG THEN
arrButtons[0]:= (xPG OR xUpDeckG)AND gvl.Current<>0;
END_IF
IF (xP1 OR xUpDeck1 OR xDownDeck1) THEN
arrButtons[1]:= (xP1 OR xUpDeck1 OR xDownDeck1) AND gvl.Current<>1;
END_IF
IF (xP2 OR xUpDeck2 OR xDownDeck2) THEN
arrButtons[2]:= (xP2 OR xUpDeck2 OR xDownDeck2) AND gvl.Current<>2;
END_IF
IF (xP3 OR xUpDeck3 OR xDownDeck3) THEN
arrButtons[3]:= (xP3 OR xUpDeck3 OR xDownDeck3) AND gvl.Current<>3;
END_IF
IF (xP4 OR xUpDeck4 OR xDownDeck4) THEN
arrButtons[4]:= (xP4 OR xUpDeck4 OR xDownDeck4) AND gvl.Current<>4;
END_IF
IF (xP5 OR xUpDeck5 OR xDownDeck5) THEN
arrButtons[5]:= (xP5 OR xUpDeck5 OR xDownDeck5) AND gvl.Current<>5;
END_IF
IF (xP6 OR xUpDeck6 OR xDownDeck6) THEN
arrButtons[6]:= (xP6 OR xUpDeck6 OR xDownDeck6) AND gvl.Current<>6;
END_IF
IF (xP7 OR xDownDeck7) THEN
arrButtons[7]:= (xP7 OR xDownDeck7) AND gvl.Current<>7;
END_IF

FOR z:= 0 TO 7 DO
	IF arrbuttons[z]=1 THEN
		//accensione luci pulsanti
		//se un certo pulsante è chiamato accendi la relativa luce
		
//pulsanti pannello interno
		IF xPG = 1 THEN xPGVis := 1; END_IF
		IF xP1 = 1 THEN xP1Vis := 1; END_IF
		IF xP2 = 1 THEN xP2Vis := 1; END_IF
		IF xP3 = 1 THEN xP3Vis := 1; END_IF
		IF xP4 = 1 THEN xP4Vis := 1; END_IF
		IF xP5 = 1 THEN xP5Vis := 1; END_IF
		IF xP6 = 1 THEN xP6Vis := 1; END_IF
		IF xP7 = 1 THEN xP7Vis := 1; END_IF
//pulsanti UpDeck
		IF xUpDeckG = 1 THEN xUpDeckGVis := 1; END_IF
		IF xUpDeck1 = 1 THEN xUpDeck1Vis := 1; END_IF
		IF xUpDeck2 = 1 THEN xUpDeck2Vis := 1; END_IF
		IF xUpDeck3 = 1 THEN xUpDeck3Vis := 1; END_IF
		IF xUpDeck4 = 1 THEN xUpDeck4Vis := 1; END_IF
		IF xUpDeck5 = 1 THEN xUpDeck5Vis := 1; END_IF
		IF xUpDeck6 = 1 THEN xUpDeck6Vis := 1; END_IF
//pulsanti DownDeck
		IF xDownDeck1 = 1 THEN xDownDeck1Vis := 1; END_IF
		IF xDownDeck2 = 1 THEN xDownDeck2Vis := 1; END_IF
		IF xDownDeck3 = 1 THEN xDownDeck3Vis := 1; END_IF
		IF xDownDeck4 = 1 THEN xDownDeck4Vis := 1; END_IF
		IF xDownDeck5 = 1 THEN xDownDeck5Vis := 1; END_IF
		IF xDownDeck6 = 1 THEN xDownDeck6Vis := 1; END_IF
		IF xDownDeck7 = 1 THEN xDownDeck7Vis := 1; END_IF
		
		//assegna le chiamate nelle destinazioni
		skip := FALSE; //inizializza skip a ogni giro
		FOR k :=0 TO 7 DO
			
			IF destinations[k]=z THEN //se c'è gia una chiamata
				arrbuttons[z]:=0;
				skip := TRUE;
			END_IF 
			
			IF (destinations[k]=-1 AND NOT skip ) THEN //AND gvl.Current<>Z
					destinations[k]:=z;	//assegna la chiamata
					EXIT;
			END_IF	
			
		END_FOR
		destination:= destinations[0];
	END_IF
END_FOR




//spegni luci
    IF iCurrentFloor = destination THEN
		CASE iCurrentFloor OF
			0:
 				xPGVis := FALSE;
				xUpDeckGVis := FALSE;
  			1:  
        		xP1Vis := FALSE;       
        		xUpDeck1Vis := FALSE;   
       			xDownDeck1Vis := FALSE;
			2:  
        		xP2Vis := FALSE;       
        		xUpDeck2Vis := FALSE;   
       			xDownDeck2Vis := FALSE;
			3:  
        		xP3Vis := FALSE;       
        		xUpDeck3Vis := FALSE;   
       			xDownDeck3Vis := FALSE;
			4:  
        		xP4Vis := FALSE;       
        		xUpDeck4Vis := FALSE;   
       			xDownDeck4Vis := FALSE;
			5:  
        		xP5Vis := FALSE;       
        		xUpDeck5Vis := FALSE;   
       			xDownDeck5Vis := FALSE;
			6:  
        		xP6Vis := FALSE;       
        		xUpDeck6Vis := FALSE;   
       			xDownDeck6Vis := FALSE;
			7:  
        		xP7Vis := FALSE;        
       			xDownDeck7Vis := FALSE;		
		END_CASE
		
		FOR w := 0 TO 6 DO
        	Destinations[w] := Destinations[w + 1];
    	END_FOR;
		
		destinations[7]:=-1;		
    END_IF
			destination:=destinations[0];
END_ACTION

ACTION _aInit_active:
State:=S_init;
destination:=-1;
FOR y:=0 TO 7 DO
	Destinations[y] := -1; 
END_FOR
END_ACTION

ACTION _aReady_active_1:
State:=S_ready;
END_ACTION

ACTION _aReady_exit_1:
state:=S_busy;
END_ACTION

END_FUNCTION_BLOCK

// Device/Application/PLC_Program
PROGRAM PLC_Program
VAR
	OpOk: BOOL;
	OpOkDest: BOOL;
END_VAR

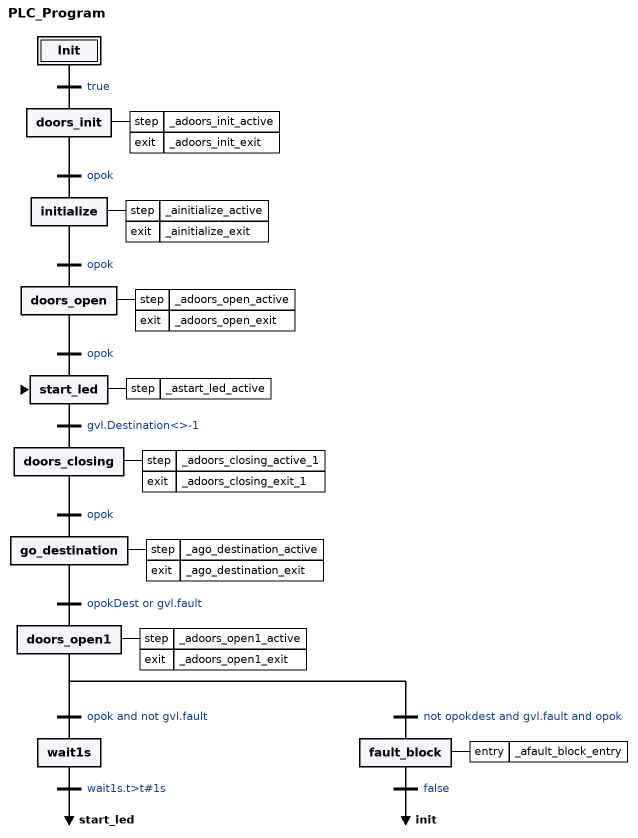
INITIAL_STEP Init:
END_STEP
TRANSITION FROM Init TO doors_init
    := true;
END_TRANSITION
STEP doors_init:
    _adoors_init_active(N);  // step action
    _adoors_init_exit(P0);  // exit action
END_STEP
TRANSITION FROM doors_init TO initialize
    := opok;
END_TRANSITION
STEP initialize:
    _ainitialize_active(N);  // step action
    _ainitialize_exit(P0);  // exit action
END_STEP
TRANSITION FROM initialize TO doors_open
    := opok;
END_TRANSITION
STEP doors_open:
    _adoors_open_active(N);  // step action
    _adoors_open_exit(P0);  // exit action
END_STEP
TRANSITION FROM doors_open TO start_led
    := opok;
END_TRANSITION
STEP start_led:
    _astart_led_active(N);  // step action
END_STEP
TRANSITION FROM start_led TO doors_closing
    := gvl.Destination<>-1;
END_TRANSITION
STEP doors_closing:
    _adoors_closing_active_1(N);  // step action
    _adoors_closing_exit_1(P0);  // exit action
END_STEP
TRANSITION FROM doors_closing TO go_destination
    := opok;
END_TRANSITION
STEP go_destination:
    _ago_destination_active(N);  // step action
    _ago_destination_exit(P0);  // exit action
END_STEP
TRANSITION FROM go_destination TO doors_open1
    := opokDest or gvl.fault;
END_TRANSITION
STEP doors_open1:
    _adoors_open1_active(N);  // step action
    _adoors_open1_exit(P0);  // exit action
END_STEP
TRANSITION FROM doors_open1 TO wait1s
    := opok and not gvl.fault;
END_TRANSITION
STEP wait1s:
END_STEP
TRANSITION FROM wait1s TO start_led
    := wait1s.t>t#1s;
END_TRANSITION
TRANSITION FROM doors_open1 TO fault_block
    := not opokdest and gvl.fault and opok;
END_TRANSITION
STEP fault_block:
    _afault_block_entry(P1);  // entry action
END_STEP
TRANSITION FROM fault_block TO init
    := false;
END_TRANSITION

ACTION _astart_led_active:
IF gvl.leds_0.State= S_ready THEN
	gvl.leds_0.Start:=TRUE;
	gvl.leds_0.Stop:=FALSE;
	END_IF
END_ACTION

ACTION _ainitialize_active:
CASE GVL.state_action OF
	
	start_action: IF gvl.motor_0.State= S_ready THEN
	gvl.motor_0.Do_:=TRUE;
	gvl.motor_0.DoWhat:=dowhats.Initialize;
	gvl.state_action:=wait_comp;
	END_IF
	
	Wait_comp: IF gvl.motor_0.done=TRUE AND gvl.motor_0.state=S_busy THEN
	gvl.motor_0.do_:=FALSE;
	gvl.state_action:=setopOK;
	END_IF
	
	SetOpOk: IF gvl.motor_0.done=FALSE THEN
	OpOk:=TRUE;// internal boolean variable	
	END_IF
	
	
END_CASE

gvl.fault:=FALSE;
END_ACTION

ACTION _ainitialize_exit:
opok:=FALSE;
gvl.state_action:=start_action;
END_ACTION

ACTION _ago_destination_active:
CASE GVL.state_action OF
	
	start_action: IF gvl.motor_0.State= S_ready THEN
	gvl.motor_0.Do_:=TRUE;
	gvl.motor_0.DoWhat:=gotodestination;
	gvl.state_action:=wait_comp;
	END_IF
	
	Wait_comp: IF gvl.motor_0.done=TRUE AND gvl.motor_0.state=S_busy AND gvl.motor_0.state<>S_faulty THEN
	gvl.motor_0.do_:=FALSE;
	gvl.state_action:=setopOK;
	END_IF
	IF gvl.motor_0.done=TRUE AND gvl.motor_0.state<>S_busy AND gvl.motor_0.state=S_faulty THEN
		GVL.fault:=TRUE;
	END_IF
	
	
	SetOpOk: IF gvl.motor_0.done=FALSE THEN
	OpOkDest:=TRUE;// internal boolean variable	
	
	END_IF
	
	
END_CASE
END_ACTION

ACTION _ago_destination_exit:
OpOk:=FALSE;
gvl.state_action:=start_action;
END_ACTION

ACTION _adoors_init_active:
CASE GVL.state_action OF
	
	start_action: IF gvl.door_opener_0.State= S_ready THEN
	gvl.door_opener_0.Do_:=TRUE;
	gvl.door_opener_0.DoWhat:=door_closing;
	gvl.state_action:=wait_comp;
	END_IF
	
	Wait_comp: IF gvl.door_opener_0.done=TRUE AND gvl.door_opener_0.state=S_busy THEN
	gvl.door_opener_0.do_:=FALSE;
	gvl.state_action:=setopOK;
	END_IF
	
	SetOpOk: IF gvl.door_opener_0.done=FALSE THEN
	OpOk:=TRUE;// internal boolean variable	
	END_IF
	
	
END_CASE
END_ACTION

ACTION _adoors_open_active:
CASE GVL.state_action OF
	
	start_action: IF gvl.door_opener_0.State= S_ready THEN
	gvl.door_opener_0.Do_:=TRUE;
	gvl.door_opener_0.DoWhat:=door_opening;
	gvl.state_action:=wait_comp;
	END_IF
	
	Wait_comp: IF gvl.door_opener_0.done=TRUE AND gvl.door_opener_0.state=S_busy THEN
	gvl.door_opener_0.do_:=FALSE;
	gvl.state_action:=setopOK;
	END_IF
	
	SetOpOk: IF gvl.door_opener_0.done=FALSE THEN
	OpOk:=TRUE;// internal boolean variable	
	END_IF
	
	
END_CASE
END_ACTION

ACTION _adoors_init_exit:
opok:=FALSE;
gvl.state_action:=start_action;
END_ACTION

ACTION _adoors_open_exit:
opok:=FALSE;
gvl.state_action:=start_action;
END_ACTION

ACTION _adoors_open1_active:
CASE GVL.state_action OF
	
	start_action: IF gvl.door_opener_0.State= S_ready THEN
	gvl.door_opener_0.Do_:=TRUE;
	gvl.door_opener_0.DoWhat:=door_opening;
	gvl.state_action:=wait_comp;
	END_IF
	
	Wait_comp: IF gvl.door_opener_0.done=TRUE AND gvl.door_opener_0.state=S_busy THEN
	gvl.door_opener_0.do_:=FALSE;
	gvl.state_action:=setopOK;
	END_IF
	
	SetOpOk: IF gvl.door_opener_0.done=FALSE THEN
	OpOk:=TRUE;// internal boolean variable	
	END_IF
	
	
END_CASE
END_ACTION

ACTION _adoors_open1_exit:
opok:=FALSE;
gvl.state_action:=start_action;
END_ACTION

ACTION _adoors_closing_exit_1:
opok:=FALSE;
gvl.state_action:=start_action;
opokdest:=false;
END_ACTION

ACTION _adoors_closing_active_1:
CASE GVL.state_action OF
	
	start_action: IF gvl.door_opener_0.State= S_ready THEN
	gvl.door_opener_0.Do_:=TRUE;
	gvl.door_opener_0.DoWhat:=door_closing;
	gvl.state_action:=wait_comp;
	END_IF
	
	Wait_comp: IF gvl.door_opener_0.done=TRUE AND gvl.door_opener_0.state=S_busy THEN
	gvl.door_opener_0.do_:=FALSE;
	gvl.state_action:=setopOK;
	END_IF
	
	SetOpOk: IF gvl.door_opener_0.done=FALSE THEN
	OpOk:=TRUE;// internal boolean variable	
	END_IF
	
	
END_CASE
END_ACTION

ACTION _afault_block_entry:
IF gvl.leds_0.State= S_busy THEN
	gvl.leds_0.Start:=FALSE;
	gvl.leds_0.Stop:=TRUE;
	END_IF
END_ACTION

END_PROGRAM

// Device/Application/Visualization
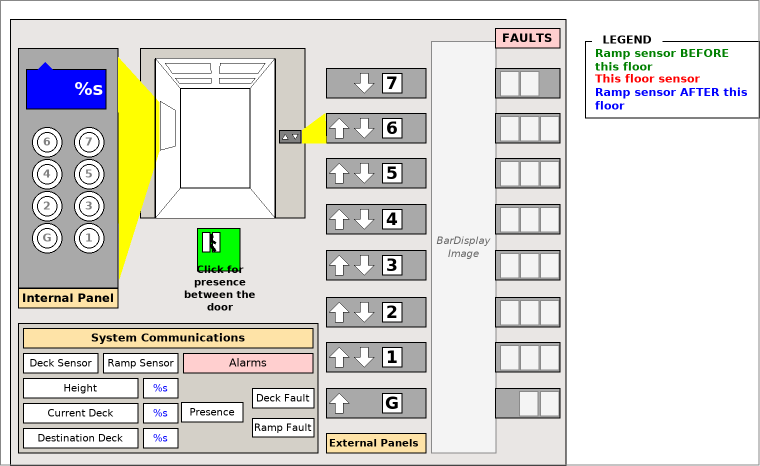
VISUALIZATION Visualization  // 760x466
    Rectangle (10,19 556x447)
    Rectangle (197,228 43x43), colour toggle: GVL.Presence
    Rectangle (18,323 300x130)
    Rectangle (326,433 100x20), "External Panels"
    Rectangle (326,342 100x30)
    Rectangle (382,347 20x20), "1"
    Polygon (354,357) (360,357) (360,347) (368,347) (368,357) (374,357) (364,367), colour toggle: GVL.DownDeck1Vis
        tap GVL.DownDeck1
    Polygon (329,357) (335,357) (335,367) (343,367) (343,357) (349,357) (339,347), colour toggle: GVL.UpDeck1Vis
        tap GVL.UpDeck1
    Rectangle (326,297 100x30)
    Rectangle (382,302 20x20), "2"
    Polygon (354,312) (360,312) (360,302) (368,302) (368,312) (374,312) (364,322), colour toggle: GVL.DownDeck2Vis
        tap GVL.DownDeck2
    Polygon (329,312) (335,312) (335,322) (343,322) (343,312) (349,312) (339,302), colour toggle: GVL.UpDeck2Vis
        tap GVL.UpDeck2
    Rectangle (326,250 100x30)
    Rectangle (382,255 20x20), "3"
    Polygon (354,265) (360,265) (360,255) (368,255) (368,265) (374,265) (364,275), colour toggle: GVL.DownDeck3Vis
        tap GVL.DownDeck3
    Polygon (329,265) (335,265) (335,275) (343,275) (343,265) (349,265) (339,255), colour toggle: GVL.UpDeck3Vis
        tap GVL.UpDeck3
    Rectangle (326,204 100x30)
    Rectangle (382,209 20x20), "4"
    Polygon (354,219) (360,219) (360,209) (368,209) (368,219) (374,219) (364,229), colour toggle: GVL.DownDeck4Vis
        tap GVL.DownDeck4
    Polygon (329,219) (335,219) (335,229) (343,229) (343,219) (349,219) (339,209), colour toggle: GVL.UpDeck4Vis
        tap GVL.UpDeck4
    Rectangle (326,158 100x30)
    Rectangle (382,163 20x20), "5"
    Polygon (354,173) (360,173) (360,163) (368,163) (368,173) (374,173) (364,183), colour toggle: GVL.DownDeck5Vis
        tap GVL.DownDeck5
    Polygon (329,173) (335,173) (335,183) (343,183) (343,173) (349,173) (339,163), colour toggle: GVL.UpDeck5Vis
        tap GVL.UpDeck5
    Rectangle (326,113 100x30)
    Rectangle (382,118 20x20), "6"
    Polygon (354,128) (360,128) (360,118) (368,118) (368,128) (374,128) (364,138), colour toggle: GVL.DownDeck6Vis
        tap GVL.DownDeck6
    Polygon (329,128) (335,128) (335,138) (343,138) (343,128) (349,128) (339,118), colour toggle: GVL.UpDeck6Vis
        tap GVL.UpDeck6
    Rectangle (326,68 100x30)
    Rectangle (382,73 20x20), "7"
    Polygon (354,83) (360,83) (360,73) (368,73) (368,83) (374,83) (364,93), colour toggle: GVL.DownDeck7Vis
        tap GVL.DownDeck7
    Rectangle (326,388 100x30)
    Rectangle (382,393 20x20), "G"
    Polygon (329,403) (335,403) (335,413) (343,413) (343,403) (349,403) (339,393), colour toggle: GVL.UpDeckGVis
        tap GVL.UpDeckG
    RoundedRectangle (18,48 100x240)
    Rectangle (18,288 100x20), "Internal Panel"
    Ellipse (74,223 30x30), colour toggle: GVL.P1Vis
    Ellipse (79,228 20x20), "1"
        tap GVL.P1
    Ellipse (32,223 30x30), colour toggle: GVL.PGVis
    Ellipse (37,228 20x20), "G"
        tap GVL.PG
    Ellipse (74,191 30x30), colour toggle: GVL.P3Vis
    Ellipse (79,196 20x20), "3"
        tap GVL.P3
    Ellipse (32,191 30x30), colour toggle: GVL.P2Vis
    Ellipse (37,196 20x20), "2"
        tap GVL.P2
    Ellipse (74,159 30x30), colour toggle: GVL.P5Vis
    Ellipse (79,164 20x20), "5"
        tap GVL.P5
    Ellipse (32,159 30x30), colour toggle: GVL.P4Vis
    Ellipse (37,164 20x20), "4"
        tap GVL.P4
    Ellipse (74,127 30x30), colour toggle: GVL.P7Vis
    Ellipse (79,132 20x20), "7"
        tap GVL.P7
    Ellipse (32,127 30x30), colour toggle: GVL.P6Vis
    Ellipse (37,132 20x20), "6"
        tap GVL.P6
    Rectangle (26,69 80x40), "%s", text variable: GVL.Destination
    Polygon (35,72) (45,62) (55,72), colour toggle: GVL.Motor_on AND GVL.Up
    Polygon (35,80) (45,90) (55,80), colour toggle: GVL.Motor_on AND NOT GVL.Up
    Group (140,48 165x170)
        Rectangle (0,0 165x170)
        Rectangle (15,10 120x160)
        Polygon (40,40) (15,10) (135,10) (110,40)
        Rectangle (40,40 70x100)
        Polygon (15,170) (40,140) (110,140) (135,170)
        Polygon (20,102) (20,53) (35,62) (35,98)
        Polygon (79,35) (79,30) (115,30) (111,35)
        Polygon (39,35) (35,30) (71,30) (71,35)
        Polygon (32,25) (25,15) (70,15) (71,25)
        Polygon (79,25) (80,15) (125,15) (118,25)
        Group (139,82 22x13)
            Rectangle (0,0 22x13)
            Polygon (3,9) (6,4) (9,9)
            Polygon (13,4) (16,9) (19,4)
    BarDisplayImage (431,41 65x412), value: GVL.Height, style: BarDisplayImage-Gray, scale format: %.0f, scale -20..160
        p3451962224: VisuNativeControl.IP_Offline.Browser
    Rectangle (495,68 65x30)
    Rectangle (495,342 65x30)
    Rectangle (495,297 65x30)
    Rectangle (495,250 65x30)
    Rectangle (495,204 65x30)
    Rectangle (495,158 65x30)
    Rectangle (495,113 65x30)
    Rectangle (495,388 65x30)
    RockerSwitch (500,345 19x25), variable: GVL.Ramp1Down, behaviour: TOGGLE, style: Switch-RockerSwitch-Green
    RockerSwitch (520,345 19x25), variable: GVL.Sensor1, behaviour: TOGGLE, style: Switch-RockerSwitch-Red
    RockerSwitch (540,345 19x25), variable: GVL.Ramp1Up, behaviour: TOGGLE, style: Switch-RockerSwitch-Blue
    RockerSwitch (500,300 19x25), variable: GVL.Ramp2Down, behaviour: TOGGLE, style: Switch-RockerSwitch-Green
    RockerSwitch (520,300 19x25), variable: GVL.Sensor2, behaviour: TOGGLE, style: Switch-RockerSwitch-Red
    RockerSwitch (540,300 19x25), variable: GVL.Ramp2Up, behaviour: TOGGLE, style: Switch-RockerSwitch-Blue
    RockerSwitch (500,253 19x25), variable: GVL.Ramp3Down, behaviour: TOGGLE, style: Switch-RockerSwitch-Green
    RockerSwitch (520,253 19x25), variable: GVL.Sensor3, behaviour: TOGGLE, style: Switch-RockerSwitch-Red
    RockerSwitch (540,253 19x25), variable: GVL.Ramp3Up, behaviour: TOGGLE, style: Switch-RockerSwitch-Blue
    RockerSwitch (500,207 19x25), variable: GVL.Ramp4Down, behaviour: TOGGLE, style: Switch-RockerSwitch-Green
    RockerSwitch (520,207 19x25), variable: GVL.Sensor4, behaviour: TOGGLE, style: Switch-RockerSwitch-Red
    RockerSwitch (540,207 19x25), variable: GVL.Ramp4Up, behaviour: TOGGLE, style: Switch-RockerSwitch-Blue
    RockerSwitch (500,161 19x25), variable: GVL.Ramp5Down, behaviour: TOGGLE, style: Switch-RockerSwitch-Green
    RockerSwitch (520,161 19x25), variable: GVL.Sensor5, behaviour: TOGGLE, style: Switch-RockerSwitch-Red
    RockerSwitch (540,161 19x25), variable: GVL.Ramp5Up, behaviour: TOGGLE, style: Switch-RockerSwitch-Blue
    RockerSwitch (500,116 19x25), variable: GVL.Ramp6Down, behaviour: TOGGLE, style: Switch-RockerSwitch-Green
    RockerSwitch (520,116 19x25), variable: GVL.Sensor6, behaviour: TOGGLE, style: Switch-RockerSwitch-Red
    RockerSwitch (540,116 19x25), variable: GVL.Ramp6Up, behaviour: TOGGLE, style: Switch-RockerSwitch-Blue
    RockerSwitch (500,71 19x25), variable: GVL.Ramp7Down, behaviour: TOGGLE, style: Switch-RockerSwitch-Green
    RockerSwitch (520,71 19x25), variable: GVL.Sensor7, behaviour: TOGGLE, style: Switch-RockerSwitch-Red
    RockerSwitch (519,391 19x25), variable: GVL.SensorG, behaviour: TOGGLE, style: Switch-RockerSwitch-Red
    RockerSwitch (540,391 19x25), variable: GVL.RampGUp, behaviour: TOGGLE, style: Switch-RockerSwitch-Blue
    Rectangle (495,28 65x20), "FAULTS"
    Polygon (302,130) (325,113) (326,143) (302,143), invisible if: (GVL.Closing OR GVL.Opening) OR GVL.Closed
    Polygon (118,57) (159,102) (159,151) (119,279), invisible if: (GVL.Closing OR GVL.Opening) OR GVL.Closed
    Rectangle (155,58 0x160)
        p3528305787: GVL.Door
    Rectangle (275,58 0x160)
        p3528305787: -GVL.Door
    Rectangle (23,328 290x20), "System Communications"
    Rectangle (183,353 130x20), "Alarms"
    Rectangle (23,353 75x20), "Deck Sensor", colour toggle: GVL.DeckSensor
    Rectangle (143,378 35x20), "%s", text variable: GVL.Height
    Rectangle (181,402 62x20), "Presence", colour toggle: GVL.Presence
    Rectangle (103,353 75x20), "Ramp Sensor", colour toggle: GVL.RampSensor
    Rectangle (143,403 35x20), "%s", text variable: GVL.Current
    Rectangle (143,428 35x20), "%s", text variable: GVL.Destination
    Rectangle (252,388 62x20), "Deck Fault", colour toggle: GVL.FaultSensorAlarm
    Rectangle (252,418 62x19), "Ramp Fault", colour toggle: GVL.FaultRampAlarm
    Rectangle (23,378 115x20), "Height"
    Rectangle (23,403 115x20), "Current Deck"
    Rectangle (23,428 115x20), "Destination Deck"
    Group (585,25 175x93)
        Rectangle (0,16 175x77)
        Rectangle (7,39 160x30), "This floor sensor"
        Rectangle (7,59 160x30), "Ramp sensor AFTER this floor"
        Rectangle (7,0 70x30), "LEGEND"
        Rectangle (7,20 160x30), "Ramp sensor BEFORE this floor"
    Group (202,232 33x34)
        toggle GVL.Presence
        Rectangle (10,0 8x20)
        Polygon (5,10) (12,20) (14,18) (5,6)
        Ellipse (6,2 5x5)
        Polygon (4,8) (13,12) (14,10) (4,4)
        Rectangle (0,0 8x20)
    Rectangle (169,273 102x31), "Click for presence between the door"
END_VISUALIZATION
